VAR_GLOBAL // INPUTS
    ivar_x AT %I*: BOOL;
END_VAR

(* stored: ProductVersion 3.1.0.18, Version 1.1.0.1 *)
